FUNCTION_BLOCK FB_BoolBindingReadOnly IMPLEMENTS I_BoolBindable
VAR
	ref : REFERENCE TO BOOL;
END_VAR

METHOD Bind
VAR_INPUT
	boolean : REFERENCE TO BOOL;
END_VAR
ref ref= boolean;
END_METHOD

{attribute 'monitoring' := 'call'}
PROPERTY IsBinded : BOOL
GET
IsBinded := __ISVALIDREF(ref);
END_GET
END_PROPERTY

{attribute 'monitoring' := 'call'}
PROPERTY Value : BOOL
GET
Value := ref;
END_GET
END_PROPERTY

END_FUNCTION_BLOCK

(* stored: Version 1.1.0.1
   POU FB_BoolBindingReadOnly: Id {f035c595-f3d7-4302-a6a4-0e368016167c}, SpecialFunc None
   Method Bind: Id {e983f9b6-0ab6-437c-96e5-a762d13ac396}
   Property IsBinded: Id {b98b2f4c-bef9-4cbe-8145-c6052f4c6749}
   Get Get: Id {c3ecef46-ab78-4488-800b-ef0c98e1f08e}
   Property Value: Id {be34ded7-c52a-40b6-be7d-89514242f0d3}
   Get Get: Id {c9cb8b85-06e5-474e-ad80-b0bc709ea14b} *)
